// TIA Portal V20 export
TYPE "LConSMC_typeAxisDynamics"
// Dynamikeinstellungen für unterschiedliche Betriebsmodi / Dynamic seetings for different operation modes
// stored: Access Published
   STRUCT
      stopDynamics { S7_SetPoint := 'True'} : "LConSMC_typeStopDynamics";   // [Einheit der Achse] Dynamiken zum Stoppen der Achse Wirksam wenn "enable" = FALSE oder wenn "speedMatch" = FALSE bei laufender Bahn / [Unit of the axis] Dynamics for stopping the axis Active if "enable" = FALSE or "speedMatch" = FLASE and running web
      syncDynamics { S7_SetPoint := 'True'} : "LConSMC_typeSyncDynamics";   // [Einheit der Achse] Dynamiken zum synchronisieren auf eine laufende Bahn Wirksam wenn "enable" & "speedMatch" = TRUE / [Unit of the axis] Dynamics for synchronizing to line speed Active if "enable" & "speedMatch" = TRUE
      operationDynamics { S7_SetPoint := 'True'} : "LConSMC_typeOperationDynamics";   // [Einheit der Achse] Dynamiken die im Normalbetrieb wirken (müssen größer oder gleich denen des Leitwertes sein!!) Wirksam wenn "enable" & "speedMatch" & "ctrlEnable" = TRUE / [Unit of the axis] Dynamics during normal operation Active if "enable" & "speedMatch" & "ctrlEnable" = TRUE
      jogDynamics { S7_SetPoint := 'True'} : "LConSMC_typeJogDynamics";   // [Einheit der Achse] Dynamiken zum Tippen der Achse Wirken wenn "JogPos" oder "jogNeg" = TRUE / [Unit of the axis] Dynamics for jogging the axis Active if "JogPos" or "jogNeg" = TRUE
   END_STRUCT;
END_TYPE
